FUNCTION F_GetThicknessForFilter : LREAL
VAR_INPUT
    stFilter : ST_Filter;
END_VAR
VAR
END_VAR

END_FUNCTION

(* stored: Version 1.1.0.1
   POU F_GetThicknessForFilter: Id {d0d7190a-2a5e-4d3e-8d36-de9d58d9f292}, SpecialFunc None *)
